INTERFACE ITF_ControlElement_HMI_Init_1 EXTENDS ITF_BaseControlElement, ITF_ControlElement_HMI_Connector_1

END_INTERFACE

(* stored: Version 1.1.0.1, ProductVersion 3.1.4024.15
   Itf ITF_ControlElement_HMI_Init_1: Id {5db9d721-721b-4974-8bfe-1ffa9bfd75bc} *)
